// TIA Portal V18 export
FUNCTION_BLOCK "Logica_PW"   // FB1, LAD
{ S7_Optimized_Access := 'TRUE' }
// stored: MemoryReserve 100, SetENOAutomatically false
   VAR_INPUT
      Selezione_Modalità { ExternalAccessible := 'False'; ExternalVisible := 'False'; ExternalWritable := 'False'} : Int;
      Richiesta_Lv_1 { ExternalAccessible := 'False'; ExternalVisible := 'False'; ExternalWritable := 'False'} : Bool;
      Richiesta_Lv_2 { ExternalAccessible := 'False'; ExternalVisible := 'False'; ExternalWritable := 'False'} : Bool;
      Richiesta_Lv_3 { ExternalAccessible := 'False'; ExternalVisible := 'False'; ExternalWritable := 'False'} : Bool;
      Disattiva_Abilitazioni { ExternalAccessible := 'False'; ExternalVisible := 'False'; ExternalWritable := 'False'} : Bool;
      Lunghezza_Pw { ExternalAccessible := 'False'; ExternalVisible := 'False'; ExternalWritable := 'False'} : Int;
   END_VAR
   VAR_OUTPUT
      Livello_1 { ExternalAccessible := 'False'; ExternalVisible := 'False'; ExternalWritable := 'False'} : Bool;
      Livello_2 { ExternalAccessible := 'False'; ExternalVisible := 'False'; ExternalWritable := 'False'} : Bool;
      Livello_3 { ExternalAccessible := 'False'; ExternalVisible := 'False'; ExternalWritable := 'False'} : Bool;
   END_VAR
   VAR_IN_OUT
      password_1 : Array[0..#N_Array] of UInt;
      password_2 : Array[0..#N_Array] of UInt;
      password_3 : Array[0..#N_Array] of UInt;
   END_VAR
   VAR
      Array_Input : Array[0..#N_Array] of UInt;
      Array_Linee : Array[0..#N_Array] of Bool;
      Conteggio : UInt;
      Risultato : UInt;
      Array_Memoria : Array[0..#N_Array] of Bool;
      Array_Fronti : Array[0..#N_Array] of Bool;
      Array_Fronti_Change : Array[0..#N_Array] of Bool;
      Visibilità : Bool;
      Numero : UInt;
      visibilità_Numeri : UInt;
      "Visibilità_Numeri_*" : UInt;
      "Visibilità_Numeri_°" : UInt;
      Fronte_Visibilità : Bool;
      Fronte_Richiesta_1 : Bool;
      Fronte_Richiesta_2 : Bool;
      Fronte_Richiesta_3 : Bool;
      Attiva_Change : Bool;
      Stato_Cambio_Pw : UInt;
      Richiesta_Lv1 : Bool;
      Richiesta_Lv2 : Bool;
      Richiesta_Lv3 : Bool;
      Fronte_Disabilità : Bool;
      Variabili_Scritte_Change : String;
      Change_Status : UInt;
      Fronte_Clock : Bool;
      "Password_Selected_ Change" : UInt;
      ET : Time;
   END_VAR
   VAR_TEMP
      n : Int;
   END_VAR
   VAR CONSTANT
      N_Array : Int := 15;
   END_VAR
   VAR_TEMP   // added for the SCL form of the ladder/FBD networks
      _w1 : Bool;
      _w2 : Bool;
      _w3 : Bool;
   END_VAR
BEGIN

REGION Network 1
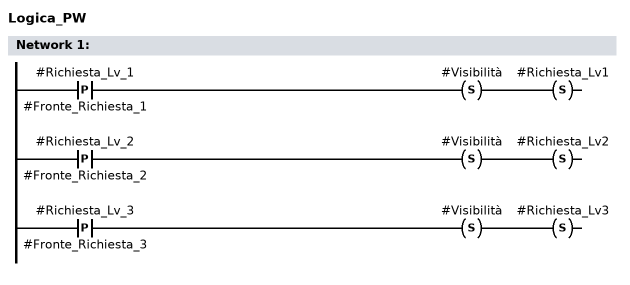
   RUNG wire#powerrail
      P_Contact(operand := #Richiesta_Lv_1, bit := #Fronte_Richiesta_1)
      S_Coil( #Visibilità )
      S_Coil( #Richiesta_Lv1 )
   END_RUNG
   RUNG wire#powerrail
      P_Contact(operand := #Richiesta_Lv_2, bit := #Fronte_Richiesta_2)
      S_Coil( #Visibilità )
      S_Coil( #Richiesta_Lv2 )
   END_RUNG
   RUNG wire#powerrail
      P_Contact(operand := #Richiesta_Lv_3, bit := #Fronte_Richiesta_3)
      S_Coil( #Visibilità )
      S_Coil( #Richiesta_Lv3 )
   END_RUNG
   // the same network as SCL:
   #_w1 := #Richiesta_Lv_1 AND NOT #Fronte_Richiesta_1;   // rising edge of #Richiesta_Lv_1
   #Fronte_Richiesta_1 := #Richiesta_Lv_1;
   IF #_w1 THEN
       #Visibilità := TRUE;
       #Richiesta_Lv1 := TRUE;
   END_IF;
   #_w2 := #Richiesta_Lv_2 AND NOT #Fronte_Richiesta_2;   // rising edge of #Richiesta_Lv_2
   #Fronte_Richiesta_2 := #Richiesta_Lv_2;
   IF #_w2 THEN
       #Visibilità := TRUE;
       #Richiesta_Lv2 := TRUE;
   END_IF;
   #_w3 := #Richiesta_Lv_3 AND NOT #Fronte_Richiesta_3;   // rising edge of #Richiesta_Lv_3
   #Fronte_Richiesta_3 := #Richiesta_Lv_3;
   IF #_w3 THEN
       #Visibilità := TRUE;
       #Richiesta_Lv3 := TRUE;
   END_IF;
END_REGION

REGION Network 2 (SCL)
   IF #Visibilità = TRUE AND #Fronte_Visibilità = false THEN
       #Variabili_Scritte_Change := 'inserisci password';
       IF #Risultato = 0 THEN  //verifico se la visibilità delle scritte è ancora a zero e nel caso la metto a 1
           #Risultato := 1;
           #visibilità_Numeri := 1;
           #Conteggio := 0;
       END_IF;
   END_IF;
   #Fronte_Visibilità := #Visibilità;
   IF #Visibilità = TRUE  THEN  //verifico se la visibilità è attiva
       REGION gestione linee e numeri/asterischi
           IF "Clock_1.25Hz" = true THEN
               #Array_Linee[#Conteggio] := true;
           ELSE
               FOR #n := 0 TO #N_Array DO
                   #Array_Linee[#n] := FALSE;
               END_FOR;
           END_IF;

           IF "Clock_10Hz" <> #Fronte_Clock THEN
               FOR #n := 0 TO #N_Array DO
                   #Array_Linee[#n] := FALSE;
               END_FOR;
           END_IF;
           #Fronte_Clock := "Clock_10Hz";


           IF #Array_Memoria[13] = true THEN
               #visibilità_Numeri := 2;
           END_IF;

           IF #Array_Memoria[13] = false & #Array_Fronti[13] = true THEN
               IF "IEC_Timer_0_DB_1".Q = true THEN
                   #visibilità_Numeri := 2;
               ELSE
                   #visibilità_Numeri := 1;
               END_IF;
           END_IF;
           #Array_Fronti[13] := #Array_Memoria[13];

           "IEC_Timer_0_DB_1".TON(IN := #Array_Memoria[13],
                                  PT := T#1s,
                                  ET => #ET);

           CASE #visibilità_Numeri OF
               1:
                   #"Visibilità_Numeri_°" := 0;
                   #"Visibilità_Numeri_*" := #Lunghezza_Pw;
               2:
                   #"Visibilità_Numeri_°" := #Lunghezza_Pw;
                   #"Visibilità_Numeri_*" := 0;
           END_CASE;
       END_REGION

       REGION rilevamento e gestione pulsanti 
           REGION rilevamento e funzionalita pulsante esc
               // pressione pulsante "ESC"
               IF (#Array_Memoria[11] = true) & (#Array_Fronti[11] = false) THEN
                   #Risultato := 1;
                   FOR #n := 0 TO #N_Array DO
                       #Array_Input[#n] := 0;
                   END_FOR;
                   FOR #n := 0 TO #N_Array DO
                       #Array_Linee[#n] := FALSE;
                   END_FOR;
                   #Conteggio := 0;
                   #Visibilità := FALSE;
                   #Richiesta_Lv1 := false;
                   #Richiesta_Lv2 := false;
                   #Richiesta_Lv3 := false;
                   #Risultato := 0;
                   #"Visibilità_Numeri_°" := 0;
                   #"Visibilità_Numeri_*" := 0;
                   #Change_Status := 0;
               END_IF;
               #Array_Fronti[11] := #Array_Memoria[11];
           END_REGION

           REGION rilevamento e funzionalità pulsante canc
               // pressione pulsante "CANC"
               IF (#Array_Memoria[12] = true) & (#Array_Fronti[12] = false) THEN
                   #Risultato := 1;
                   FOR #n := 0 TO #N_Array DO
                       #Array_Input[#n] := 0;
                   END_FOR;
                   #Conteggio := 0;
               END_IF;
               #Array_Fronti[12] := #Array_Memoria[12];
           END_REGION

           REGION rilevamento e funzionalità pulsante indietro
               // pressione pulsante indietro
               IF (#Array_Memoria[14] = true) & (#Array_Fronti[14] = false) THEN
                   IF #Conteggio > 0 THEN
                       #Conteggio := #Conteggio - 1;
                       #Array_Input[#Conteggio] := 0;
                   END_IF;
               END_IF;
               #Array_Fronti[14] := #Array_Memoria[14];
           END_REGION

           REGION rilevamento e funzionalità pulsante disattiva abilitazioni
               IF #Disattiva_Abilitazioni = true & #Fronte_Disabilità = false THEN
                   #Livello_1 := false;
                   #Livello_2 := false;
                   #Livello_3 := false;
               END_IF;
               #Fronte_Disabilità := #Disattiva_Abilitazioni;
           END_REGION
       END_REGION

       REGION rilevazione pressione pulsanti fintanto che il numero di caratteri inseriti non superi la lunghezza_pw

           IF #Conteggio < #Lunghezza_Pw THEN  //verifico se le volte in cui i numeri sono stati premuti è minore di #lunghezza_pw

               //vado a registrare gli input dei pulsanti numerici
               IF (#Array_Memoria[0] = true) & (#Array_Fronti[0] = false) THEN
                   #Array_Linee[#Numero] := FALSE;
                   #Array_Input[#Conteggio] := 0;
                   #Conteggio := #Conteggio + 1;
               END_IF;

               #Array_Fronti[0] := #Array_Memoria[0];

               IF (#Array_Memoria[1] = true) & (#Array_Fronti[1] = false) THEN
                   #Array_Linee[#Numero] := FALSE;
                   #Array_Input[#Conteggio] := 1;
                   #Conteggio := #Conteggio + 1;
               END_IF;
               #Array_Fronti[1] := #Array_Memoria[1];

               IF (#Array_Memoria[2] = true) & (#Array_Fronti[2] = false) THEN
                   #Array_Linee[#Numero] := FALSE;
                   #Array_Input[#Conteggio] := 2;
                   #Conteggio := #Conteggio + 1;
               END_IF;
               #Array_Fronti[2] := #Array_Memoria[2];

               IF (#Array_Memoria[3] = true) & (#Array_Fronti[3] = false) THEN
                   #Array_Linee[#Numero] := FALSE;
                   #Array_Input[#Conteggio] := 3;
                   #Conteggio := #Conteggio + 1;
               END_IF;
               #Array_Fronti[3] := #Array_Memoria[3];

               IF (#Array_Memoria[4] = true) & (#Array_Fronti[4] = false) THEN
                   #Array_Linee[#Numero] := FALSE;
                   #Array_Input[#Conteggio] := 4;
                   #Conteggio := #Conteggio + 1;
               END_IF;
               #Array_Fronti[4] := #Array_Memoria[4];

               IF (#Array_Memoria[5] = true) & (#Array_Fronti[5] = false) THEN
                   #Array_Linee[#Numero] := FALSE;
                   #Array_Input[#Conteggio] := 5;
                   #Conteggio := #Conteggio + 1;
               END_IF;
               #Array_Fronti[5] := #Array_Memoria[5];

               IF (#Array_Memoria[6] = true) & (#Array_Fronti[6] = false) THEN
                   #Array_Linee[#Numero] := FALSE;
                   #Array_Input[#Conteggio] := 6;
                   #Conteggio := #Conteggio + 1;
               END_IF;
               #Array_Fronti[6] := #Array_Memoria[6];

               IF (#Array_Memoria[7] = true) & (#Array_Fronti[7] = false) THEN
                   #Array_Linee[#Numero] := FALSE;
                   #Array_Input[#Conteggio] := 7;
                   #Conteggio := #Conteggio + 1;
               END_IF;
               #Array_Fronti[7] := #Array_Memoria[7];

               IF (#Array_Memoria[8] = true) & (#Array_Fronti[8] = false) THEN
                   #Array_Linee[#Numero] := FALSE;
                   #Array_Input[#Conteggio] := 8;
                   #Conteggio := #Conteggio + 1;
               END_IF;
               #Array_Fronti[8] := #Array_Memoria[8];

               IF (#Array_Memoria[9] = true) & (#Array_Fronti[9] = false) THEN
                   #Array_Linee[#Numero] := FALSE;
                   #Array_Input[#Conteggio] := 9;
                   #Conteggio := #Conteggio + 1;
               END_IF;
               #Array_Fronti[9] := #Array_Memoria[9];
           END_IF;
       END_REGION

       REGION Change_Status=0
           IF #Change_Status = 0 THEN

               REGION Restituzione risultato in base alla MODalità di funzionamento selezionata

                   IF (#Array_Memoria[10] = true) & (#Array_Fronti[10] = false) THEN
                       CASE #Selezione_Modalità OF
                           0:
                               IF #Array_Input = #password_1 THEN
                                   #Risultato := 2;
                                   #Livello_1 := true;
                                   #Livello_2 := true;
                                   #Livello_3 := true;
                                   #Variabili_Scritte_Change := 'Password corretta';
                               ELSE
                                   IF #Array_Input = #password_2 THEN
                                       #Risultato := 2;
                                       #Livello_2 := true;
                                       #Livello_3 := true;
                                       #Variabili_Scritte_Change := 'Password corretta';
                                   ELSE
                                       IF #Array_Input = #password_3 THEN
                                           #Risultato := 2;
                                           #Livello_3 := true;
                                           #Variabili_Scritte_Change := 'Password corretta';
                                       ELSE
                                           #Risultato := 3;
                                           #Variabili_Scritte_Change := 'Password sbagliata';
                                       END_IF;
                                   END_IF;
                               END_IF;
                           1:
                               IF #Richiesta_Lv1 = true THEN
                                   IF #Array_Input = #password_1 THEN
                                       #Risultato:= 2;
                                       #Livello_1 := true;
                                   ELSE
                                       #Risultato := 3;
                                   END_IF;
                               END_IF;
                               IF #Richiesta_Lv2 = true THEN
                                   IF #Array_Input = #password_2 THEN
                                       #Risultato := 2;
                                       #Livello_2 := true;
                                   ELSE
                                     #Risultato := 3;
                                   END_IF;
                               END_IF;
                               IF #Richiesta_Lv3 = true THEN
                                   IF #Array_Input = #password_3 THEN
                                       #Risultato := 2;
                                       #Livello_3 := true;
                                   ELSE
                                       #Risultato := 3;
                                   END_IF;
                               END_IF;
                           2:
                               IF #Array_Input = #password_1 THEN
                                  #Risultato := 2;
                                   #Livello_1:= true;
                                   #Livello_2:= true;
                                   #Livello_3 := true;
                               ELSE
                                   #Risultato := 3;
                               END_IF;
                       END_CASE;
                   END_IF;
                   #Array_Fronti[10] := #Array_Memoria[10];

               END_REGION

           END_IF;

       END_REGION

       REGION gestione modalità cambio password

           REGION Pressione pulsante change password ed entrata nella modalità sovrascrittura
               IF (#Array_Memoria[15] = true) & (#Array_Fronti[15] = false) THEN
                   #Variabili_Scritte_Change := 'Seleziona password da modificare';
                   FOR #n := 0 TO #N_Array DO
                       #Array_Input[#n] := 0;
                   END_FOR;
                   #Conteggio := 0;
                   #Change_Status := 1;
               END_IF;
               #Array_Fronti[15] := #Array_Memoria[15];
           END_REGION

           REGION Change_Status=1

               IF #Change_Status = 1 THEN
                   IF (#Array_Memoria[1] = true) & (#Array_Fronti_Change[1] = false) THEN
                       FOR #n := 0 TO #N_Array DO
                           #Array_Input[#n] := 0;
                       END_FOR;
                       #Conteggio := 0;
                       #Variabili_Scritte_Change := 'password precedente';
                       #Change_Status := 2;
                       #"Password_Selected_ Change" := 1;
                   END_IF;
                   #Array_Fronti_Change[1] := #Array_Memoria[1];

                   IF (#Array_Memoria[2] = true) & (#Array_Fronti_Change[2] = false) THEN
                       FOR #n := 0 TO #N_Array DO
                           #Array_Input[#n] := 0;
                       END_FOR;
                       #Conteggio := 0;
                       #Variabili_Scritte_Change :='password precedente'; // 
                       #Change_Status := 2;
                       #"Password_Selected_ Change" := 2;
                   END_IF;
                   #Array_Fronti_Change[2] := #Array_Memoria[2];


                   IF (#Array_Memoria[3] = true) & (#Array_Fronti_Change[3] = false) THEN
                       FOR #n := 0 TO #N_Array DO
                           #Array_Input[#n] := 0;
                       END_FOR;
                       #Conteggio := 0;
                       #Variabili_Scritte_Change :='password precedente';
                       #Change_Status := 2;
                       #"Password_Selected_ Change" := 3;
                   END_IF;
                   #Array_Fronti_Change[3] := #Array_Memoria[3];
               END_IF;

           END_REGION


           REGION Change_Status=2
               IF #Change_Status = 2 THEN
                   IF #Array_Memoria[10] = true & #Array_Fronti_Change[10] = FALSE THEN
                       CASE #"Password_Selected_ Change" OF
                           1:
                               IF #Array_Input = #"password_1" THEN
                                   #Change_Status := 3;
                                   FOR #n := 0 TO #N_Array DO
                                       #Array_Input[#n] := 0;
                                   END_FOR;
                                   #Conteggio := 0;
                                   #Variabili_Scritte_Change := 'Nuova password';
                               ELSE
                                   #Variabili_Scritte_Change := 'Password errata';
                               END_IF;
                           2:
                               IF #Array_Input = #password_2 THEN
                                   #Change_Status := 3;
                                   FOR #n := 0 TO #N_Array DO
                                       #Array_Input[#n] := 0;
                                   END_FOR;
                                   #Conteggio := 0;
                                   #Variabili_Scritte_Change := 'Nuova password';
                               ELSE
                                   #Variabili_Scritte_Change := 'Password errata';
                               END_IF;
                           3:
                               IF #Array_Input = #password_3 THEN
                                   #Change_Status := 3;
                                   FOR #n := 0 TO #N_Array DO
                                       #Array_Input[#n] := 0;
                                   END_FOR;
                                   #Conteggio := 0;
                                   #Variabili_Scritte_Change := 'Nuova password';
                               ELSE
                                   #Variabili_Scritte_Change := 'Password errata';
                               END_IF;
                       END_CASE;
                   END_IF;
                   #Array_Fronti_Change[10] := #Array_Memoria[10];
               END_IF;


           END_REGION


           REGION Change_Status=3
                   IF #Change_Status = 3 THEN
                       IF #Array_Memoria[10] = true & #Array_Fronti_Change[11] = FALSE THEN
                           CASE #"Password_Selected_ Change" OF
                               1:
                                   #Variabili_Scritte_Change := 'Password modificata';
                                   #"password_1" := #Array_Input;
                                   FOR #n := 0 TO #N_Array DO
                                       #Array_Input[#n] := 0;
                                   END_FOR;
                                   #Conteggio := 0;
                                   #Change_Status := 0;

                               2:
                                   #Variabili_Scritte_Change := 'Password modificata';
                                   #"password_2" := #Array_Input;
                                   FOR #n := 0 TO #N_Array DO
                                       #Array_Input[#n] := 0;
                                   END_FOR;
                                   #Conteggio := 0;
                                   #Change_Status := 0;

                               3:
                                   #Variabili_Scritte_Change := 'Password modificata';
                                   #"password_3" := #Array_Input;
                                   FOR #n := 0 TO #N_Array DO
                                       #Array_Input[#n] := 0;
                                   END_FOR;
                                   #Conteggio := 0;
                                   #Change_Status := 0;

                           END_CASE;
                       END_IF;
                       #Array_Fronti_Change[11] := #Array_Memoria[10];
                   END_IF;


               END_REGION



       END_REGION

   END_IF;
END_REGION
END_FUNCTION_BLOCK
